FUNCTION_BLOCK SEL_ANY (* Abstract superclass for IEC 61131-3 binary Selections *)
  (* Standard: 61131-3 *)
  (* Version 0.0, 2004-12-15, JHC, Rockwell Automation, Converted from SRC format. *)
  (* Compiler header: package fb.rt.plc.select; *)
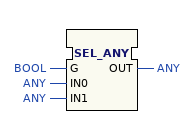
  VAR_INPUT
    G : BOOL; (* Selector *)
    IN0 : ANY; (* Selected when G=0 *)
    IN1 : ANY; (* Selected when G=1 *)
  END_VAR
  VAR_OUTPUT
    OUT : ANY; (* Selected value *)
  END_VAR
END_FUNCTION_BLOCK
